// TIA Portal V16 export
// export: Created 2024-09-05T17:39:19.6341403Z, ExportSetting WithDefaults, DisplayName Totally Integrated Automation Portal, DisplayVersion V16 Update 6, DisplayName TIA Portal Version Control Interface, DisplayVersion V16 Update 2, DisplayName TIA Portal Openness, DisplayVersion V16 Update 6, DisplayName STEP 7 Professional, DisplayVersion V16 Update 6, DisplayName STEP 7 Safety, DisplayVersion V16, DisplayName WinCC Advanced, DisplayVersion V16 Update 6
DATA_BLOCK "SystemHMI"   // DB10
{ S7_Optimized_Access := 'TRUE' }
VERSION : 0.1
// stored: AutoNumber false, DBAccessibleFromOPCUA true, IsOnlyStoredInLoadMemory false, IsRetainMemResEnabled false, IsWriteProtectedInAS false, MemoryReserve 100
   VAR
      AlarmActive : Bool := FALSE;
      AlarmActiveBlinking : Bool := FALSE;
      WarningActive : Bool := FALSE;
      BasicPosition : Bool := FALSE;
      GoToBasicPosition : Bool := FALSE;
      ManualMode : Bool := TRUE;
      AutomaticMode : Bool := FALSE;
      ManualCommand : Int := 0;
      BasicPositionMessage : Int := 0;
      BasicPositionStep : Int := 0;
      ManualFromRobot : Bool := FALSE;
      HydraulicPumpAutoControl : Bool := FALSE;
      BasicPositionSt1 : Bool := FALSE;
      BasicPositionSt2 : Bool := FALSE;
      BasicPositionFitting : Bool := FALSE;
      BasicPositionGripper1 : Bool := FALSE;
      BasicPositionStartHMI : Bool := FALSE;
      AutoStartHMI : Bool := FALSE;
      ResetPartsErrors : Bool := FALSE;
      ModeChanged : Bool := FALSE;
   END_VAR
BEGIN
END_DATA_BLOCK
